PROGRAM MAIN
VAR
	Analogwerte: Analogwerte;
END_VAR

Analogwerte();

END_PROGRAM

(* stored: Version 1.1.0.1, ProductVersion 3.1.4022.7
   POU MAIN: Id {9753ee2a-e609-4081-882e-52e8c65681cc}, SpecialFunc None *)
